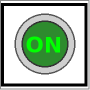
VISUALIZATION Vis_DigitalInput_1  // 90x90
VAR_IN_OUT
	stHMI_DigitalInput:stHMI_DigitalInput;
END_VAR
    Rectangle (1,3 86x83)
        p3092690914: stHMI_DigitalInput.iMode=2
    Lamp1 (10,9 70x70), style: Lamp-Lamp1-Gray
    Lamp1 (10,9 70x70), invisible if: stHMI_DigitalInput.bOn=0, style: Lamp-Lamp1-Green
    Label (16,31 56x28), "ON", invisible if: stHMI_DigitalInput.bOn=0
END_VISUALIZATION

(* stored: Version 1.1.0.1, ProductVersion 3.1.4024.11
   Visu Vis_DigitalInput_1: Id {34c9d918-78a5-4d22-b127-1e0ebf774685} *)
